// Mitsubishi GX Works2 project: 0702-2   PLC: Q02/Q02H

PROGRAM MAIN
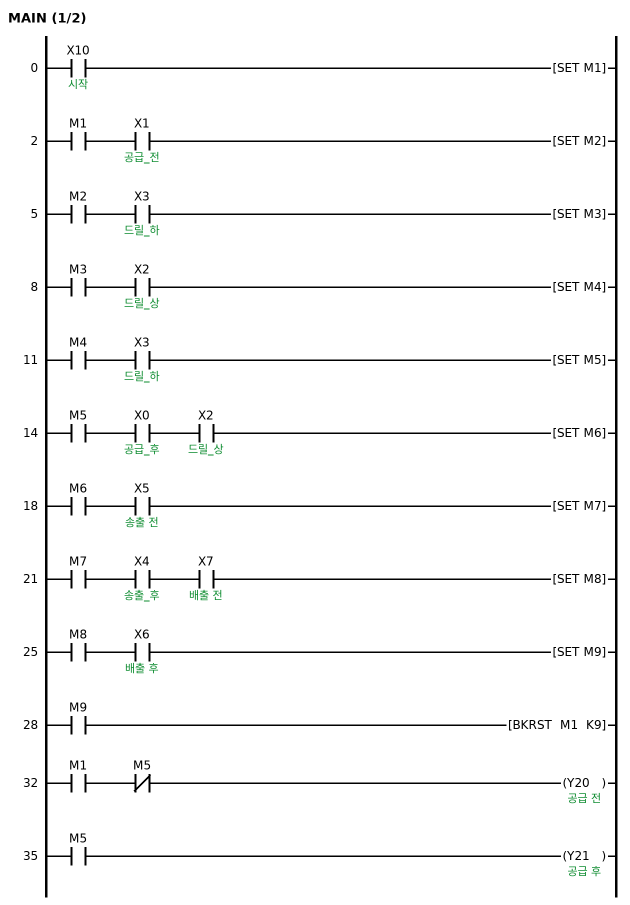
0     LD      X10  ; 시작
      SET     M1
2     LD      M1
      AND     X1  ; 공급_전
      SET     M2
5     LD      M2
      AND     X3  ; 드릴_하
      SET     M3
8     LD      M3
      AND     X2  ; 드릴_상
      SET     M4
11    LD      M4
      AND     X3  ; 드릴_하
      SET     M5
14    LD      M5
      AND     X0  ; 공급_후
      AND     X2  ; 드릴_상
      SET     M6
18    LD      M6
      AND     X5  ; 송출 전
      SET     M7
21    LD      M7
      AND     X4  ; 송출_후
      AND     X7  ; 배출 전
      SET     M8
25    LD      M8
      AND     X6  ; 배출 후
      SET     M9
28    LD      M9
      BKRST   M1 K9
32    LD      M1
      ANI     M5
      OUT     Y20  ; 공급 전
35    LD      M5
      OUT     Y21  ; 공급 후
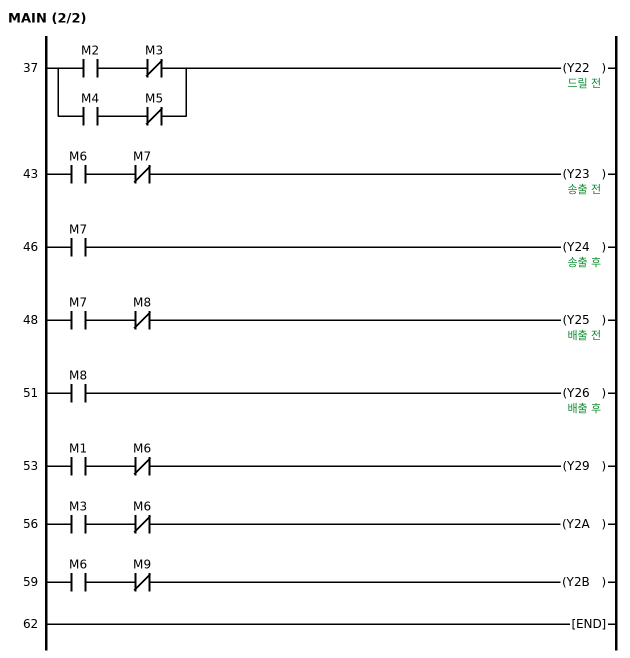
37    LD      M2
      ANI     M3
      LD      M4
      ANI     M5
      ORB
      OUT     Y22  ; 드릴 전
43    LD      M6
      ANI     M7
      OUT     Y23  ; 송출 전
46    LD      M7
      OUT     Y24  ; 송출 후
48    LD      M7
      ANI     M8
      OUT     Y25  ; 배출 전
51    LD      M8
      OUT     Y26  ; 배출 후
53    LD      M1
      ANI     M6
      OUT     Y29
56    LD      M3
      ANI     M6
      OUT     Y2A
59    LD      M6
      ANI     M9
      OUT     Y2B
62    END
END_PROGRAM

// device comments not shown above
X11  ; 정지
